VAR_GLOBAL PERSISTENT 
	

Mc:Machine;

END_VAR

(* stored: Version 1.1.0.1, ProductVersion 3.1.4024.9
   GVL Mc: Id {9bab8bad-8f58-466d-99ee-829cf0e62d22} *)
